{attribute 'qualified_only'}
{attribute 'strict'}
TYPE E_StateSequencer :
(
	OFF					:= 0,
	INIT_1				:= 10,
	INIT_2				:= 11,
	INIT_3				:= 12,
	HOMING_1			:= 90,
	HOMING_2			:= 91,
	
	IDLE				:= 100,
	OPEN_FILE			:= 110,
	CLOSE_FILE			:= 120,
	CHANGE_MATERIAL_1	:= 130,
	CHANGE_MATERIAL_2	:= 131,
	CHANGE_MATERIAL_3	:= 132,
	
	READY				:= 200,
	
	PREP_PRINTING		:= 300,
	PREP_PRINTING_HEX_1	:= 301,
	PREP_PRINTING_HEX_2	:= 302,
	PREP_PRINTING_HEX_3	:= 303,
	PREP_PRINTING_HEX_4 := 304,
	PREP_PRINTING_EXT	:= 305,
	PREP_PRINTING_HEX_5	:= 306,
	PREP_PRINTING_HEX_6	:= 307,
	PREP_PRINTING_HEX_7	:= 308,
	
	READ_FILE			:= 310,
	EXECUTE_LINE		:= 320,
	
	WRITE_KOS			:= 330,
	WRITE_FEED			:= 331,
	WRITE_PROG			:= 335,
	
	EXTRUDER_ON_1		:= 340,
	EXTRUDER_ON_2		:= 341,
	
	EXTRUDER_OFF_1		:= 350,
	START_EXTRUDING		:= 351,
	EXTRUDER_OFF_2		:= 352,
	
	STOP_EXTRUDING		:= 360,
	
	PAUSE				:= 390,
	
	ABORTED				:= 400,
	
	FINISHED			:= 500,
	
	SHUTDOWN			:= 600
);
END_TYPE

(* stored: Version 1.1.0.1
   EnumerationTextList E_StateSequencer: Id {86bc2c5b-3169-4949-a177-892e2e46c23f} *)
